// TIA Portal V16 export
// export: Created 2022-02-04T14:40:18.707467Z, ExportSetting WithDefaults, DisplayName Totally Integrated Automation Portal, DisplayVersion V16 Update 1, DisplayName TIA Portal Version Control Interface, DisplayVersion V16, DisplayName TIA Portal Openness, DisplayVersion V16, DisplayName SINAMICS Startdrive Advanced, DisplayVersion V16 Update 5, DisplayName SINAMICS Startdrive G130, G150, S120, S150, SINAMICS MV, S210, DisplayVersion V16 Update 5, DisplayName SINAMICS Startdrive G110M, G120, G120C, G120D, G120P, G115D, DisplayVersion V16 Update 5, DisplayName STEP 7 Professional, DisplayVersion V16, DisplayName STEP 7 Safety, DisplayVersion V16, DisplayName WinCC Advanced, DisplayVersion V16, DisplayName SIMATIC Visualization Architect, DisplayVersion V16
DATA_BLOCK "DGI"   // DB2
VERSION : 0.1
// stored: AutoNumber true, InstanceOfName GetDiskretInputs, InstanceOfType FB
"GetDiskretInputs"
   // VAR RETAIN
   //    K1_1122L1 : Bool;
   //    K1_113_13L1 : Bool;
   //    K1_113_24L1 : Bool;
   //    K1_113_35L1 : Bool;
   //    k1_113_46L1 : Bool;
   //    Varalla : Bool;
   //    Varalla1 : Bool;
   //    Varalla2 : Bool;
   //    F211K1_211K2 : Bool;
   //    F212K1 : Bool;
   //    F213K1 : Bool;
   //    F214K1 : Bool;
   //    Varalla3 : Bool;
   //    Varalla4 : Bool;
   //    Varalla5 : Bool;
   //    Varalla6 : Bool;
   //    F221K1 : Bool;
   //    F222K1 : Bool;
   //    F223K1 : Bool;
   //    F224K1 : Bool;
   //    F225K1 : Bool;
   //    F330K1 : Bool;
   //    Varalla8 : Bool;
   //    Varalla9 : Bool;
   //    F231K1 : Bool;
   //    F232K1 : Bool;
   //    F233K1 : Bool;
   //    F234K1 : Bool;
   //    F235K1_235K2 : Bool;
   //    Varalla10 : Bool;
   //    Varalla11 : Bool;
   //    Varalla12 : Bool;
   //    F311K1_311K2 : Bool;
   //    F312K1 : Bool;
   //    F313K1_313K2 : Bool;
   //    F314K1 : Bool;
   //    F315K1 : Bool;
   //    F316K1 : Bool;
   //    F317K1 : Bool;
   //    Varalla13 : Bool;
   //    F321K1_321K2 : Bool;
   //    F322K1_322K2 : Bool;
   //    F323K1_323K2 : Bool;
   //    F325K1 : Bool;
   //    Varalla14 : Bool;
   //    Varalla15 : Bool;
   //    Varalla16 : Bool;
   //    Varalla17 : Bool;
   //    F331K1 : Bool;
   //    F332K1 : Bool;
   //    F333K1 : Bool;
   //    F334K1 : Bool;
   //    F335K1 : Bool;
   //    F336K1 : Bool;
   //    F337K1 : Bool;
   //    K1_323U1 : Bool;
   //    K1_221U1 : Bool;
   //    K1_213U1 : Bool;
   //    K1_215U1 : Bool;
   //    K1_222U1 : Bool;
   //    K1_225U1 : Bool;
   //    K1_231U1 : Bool;
   //    K1_233U1 : Bool;
   //    K1_317U1 : Bool;
   //    K1_332U1 : Bool;
   //    K1_333U1 : Bool;
   //    K1_334U1 : Bool;
   //    K1_335U1 : Bool;
   //    K1_336U1 : Bool;
   //    K1_223U1 : Bool;
   //    K1_324U1 : Bool;
   //    K1_325U1 : Bool;
   //    K1_112_S1 : Bool;
   //    K1_112_S2 : Bool;
   //    K1_112_S3 : Bool;
   //    Varalla22 : Bool;
   //    K1_113_S11 : Bool;
   //    K1_113_S12 : Bool;
   //    k1_113_S13 : Bool;
   //    Varalla23 : Bool;
   //    Varalla24 : Bool;
   //    FC_223_1 : Bool;
   //    FC_223_2 : Bool;
   //    FC_223_3 : Bool;
   //    Varalla28 : Bool;
   //    Varalla29 : Bool;
   //    Varalla30 : Bool;
   //    Varalla31 : Bool;
   //    Liftdown : Bool;
   //    LiftUp : Bool;
   //    sloidoski : Bool;
   //    sloidoski2 : Bool;
   //    doskavpriymkeelevator : Bool;
   //    koncevik1 : Bool;
   //    koncevik2 : Bool;
   //    nakloniytransporter : Bool;
   //    FC_18_Length : Bool;
   //    F2_1m : Bool;
   //    F2_4m : Bool;
   //    F2_7m : Bool;
   //    F3_0m : Bool;
   //    F3_3m : Bool;
   //    F3_6m : Bool;
   //    F3_9m : Bool;
   //    F4_2m : Bool;
   //    F4_5m : Bool;
   //    F4_8m : Bool;
   //    F5_1m : Bool;
   //    F5_4m : Bool;
   //    F5_7m : Bool;
   //    F6_0m : Bool;
   //    PodBort_1 : Bool;
   //    PodBort_2 : Bool;
   //    "312Alarm" : Bool;
   //    S14_2 : Bool;
   //    S14_3 : Bool;
   //    B14_4 : Bool;
   //    B14_5 : Bool;
   //    K1_312U1 : Bool;
   //    S14_7 : Bool;
   //    S15_0 : Bool;
   //    S15_1 : Bool;
   //    S15_2 : Bool;
   //    reserv5 : Bool;
   //    Index : Bool;
   //    B15_5 : Bool;
   //    B15_6 : Bool;
   //    B15_7 : Bool;
   //    FC_232_1 : Bool;
   //    S16_1 : Bool;
   //    S16_2 : Bool;
   //    E16_3 : Bool;
   //    E16_4 : Bool;
   //    FC_232_2 : Bool;
   //    B16_6 : Bool;
   //    S16_7 : Bool;
   //    B17_0 : Bool;
   //    B17_1 : Bool;
   //    B17_2 : Bool;
   //    B17_3 : Bool;
   //    B17_4 : Bool;
   //    Varalla32 : Bool;
   //    Varalla33 : Bool;
   //    Varalla34 : Bool;
   //    B18_0 : Bool;
   //    B18_1 : Bool;
   //    S18_2 : Bool;
   //    S18_3 : Bool;
   //    B18_4 : Bool;
   //    B18_5 : Bool;
   //    B18_6 : Bool;
   //    B18_7 : Bool;
   //    B19_0 : Bool;
   //    Varalla35 : Bool;
   //    Varalla36 : Bool;
   //    Varalla37 : Bool;
   //    Varalla38 : Bool;
   //    Varalla39 : Bool;
   //    Varalla40 : Bool;
   //    Varalla41 : Bool;
   //    Varalla42 : Bool;
   //    Varalla43 : Bool;
   //    Varalla44 : Bool;
   //    Varalla45 : Bool;
   //    Varalla46 : Bool;
   //    Varalla47 : Bool;
   //    Varalla48 : Bool;
   //    Varalla49 : Bool;
   //    Varalla50 : Bool;
   //    Varalla51 : Bool;
   //    Varalla52 : Bool;
   //    Varalla53 : Bool;
   //    Varalla54 : Bool;
   //    Varalla55 : Bool;
   //    Varalla56 : Bool;
   //    Varalla57 : Bool;
   //    B22_0 : Bool;
   //    B22_1 : Bool;
   //    S22_2 : Bool;
   //    S22_3 : Bool;
   //    B22_4 : Bool;
   //    B22_5 : Bool;
   //    B22_6 : Bool;
   //    FC_22_7 : Bool;
   //    B23_0 : Bool;
   //    B23_1 : Bool;
   //    Varalla59 : Bool;
   //    Varalla60 : Bool;
   //    Varalla61 : Bool;
   //    Varalla62 : Bool;
   //    FC_23_6 : Bool;
   //    FC_23_7 : Bool;
   //    S76 : Bool;
   //    S76_1 : Bool;
   //    S76_2 : Bool;
   //    S76_3 : Bool;
   //    E76_4 : Bool;
   //    S76_5 : Bool;
   //    S76_6 : Bool;
   //    E76_7 : Bool;
   //    S77_0 : Bool;
   //    E77_1 : Bool;
   //    S77_2 : Bool;
   //    S77_3 : Bool;
   //    S77_4 : Bool;
   //    S77_5 : Bool;
   //    S77_6 : Bool;
   //    E77_7 : Bool;
   //    S78_0 : Bool;
   //    E78_1 : Bool;
   //    S78_2 : Bool;
   //    E78_3 : Bool;
   //    S78_4 : Bool;
   //    E78_5 : Bool;
   //    S78_6 : Bool;
   //    E78_7 : Bool;
   //    S79_0 : Bool;
   //    S79_1 : Bool;
   //    E79_2 : Bool;
   //    S79_3 : Bool;
   //    S79_4 : Bool;
   //    S79_5 : Bool;
   //    S79_6 : Bool;
   //    E79_7 : Bool;
   //    S80_0 : Bool;
   //    E80_1 : Bool;
   //    S80_2 : Bool;
   //    E80_3 : Bool;
   //    S80_4 : Bool;
   //    S80_5 : Bool;
   //    E80_6 : Bool;
   //    S80_7 : Bool;
   //    Varalla106 : Bool;
   //    Varalla107 : Bool;
   //    Varalla108 : Bool;
   //    Varalla109 : Bool;
   //    Varalla110 : Bool;
   //    Varalla111 : Bool;
   //    Varalla112 : Bool;
   //    Varalla113 : Bool;
   //    S82_0 : Bool;
   //    S81_1 : Bool;
   //    E82_2 : Bool;
   //    S82_3 : Bool;
   //    S82_4 : Bool;
   //    E82_5 : Bool;
   //    S82_6 : Bool;
   //    E82_7 : Bool;
   //    S83_0 : Bool;
   //    E83_1 : Bool;
   //    E83_2 : Bool;
   //    E83_3 : Bool;
   //    S83_4 : Bool;
   //    Varalla114 : Bool;
   //    Varalla115 : Bool;
   //    Varalla116 : Bool;
   //    S84_0 : Bool;
   //    S84_1 : Bool;
   //    E84_2 : Bool;
   //    S84_3 : Bool;
   //    S84_4 : Bool;
   //    S84_5 : Bool;
   //    E84_6 : Bool;
   //    S84_7 : Bool;
   //    E85_0 : Bool;
   //    S85_1 : Bool;
   //    E85_2 : Bool;
   //    S85_3 : Bool;
   //    E85_4 : Bool;
   //    S85_5 : Bool;
   //    E85_6 : Bool;
   //    S85_7 : Bool;
   //    S86_0 : Bool;
   //    E86_1 : Bool;
   //    S86_2 : Bool;
   //    S86_3 : Bool;
   //    S86_4 : Bool;
   //    S86_5 : Bool;
   //    Varalla117 : Bool;
   //    Varalla118 : Bool;
   //    S87_0 : Bool;
   //    S87_1 : Bool;
   //    E87_2 : Bool;
   //    S87_3 : Bool;
   //    S87_4 : Bool;
   //    Varalla119 : Bool;
   //    Varalla120 : Bool;
   //    Varalla121 : Bool;
   //    S88_0 : Bool;
   //    K3_3 : Bool;
   //    S88_2 : Bool;
   //    E88_3 : Bool;
   //    S88_4 : Bool;
   //    S88_5 : Bool;
   //    E88_6 : Bool;
   //    S88_7 : Bool;
   //    S89_0 : Bool;
   //    S89_1 : Bool;
   //    S89_2 : Bool;
   //    S89_3 : Bool;
   //    Varalla122 : Bool;
   //    Varalla123 : Bool;
   //    Varalla124 : Bool;
   //    Varalla125 : Bool;
   //    S90_0 : Bool;
   //    S90_1 : Bool;
   //    S90_2 : Bool;
   //    Varalla126 : Bool;
   //    S90_4 : Bool;
   //    E90_5 : Bool;
   //    S90_6 : Bool;
   //    E90_7 : Bool;
   //    S91_0 : Bool;
   //    E91_1 : Bool;
   //    S91_2 : Bool;
   //    Varalla127 : Bool;
   //    Varalla128 : Bool;
   //    Varalla129 : Bool;
   //    Varalla130 : Bool;
   //    Varalla131 : Bool;
   //    S214 : Bool;
   //    BrakDroper_front : Bool;
   //    BrakDroppperBob_old : Bool;
   //    UporDefectivePFM_timer : TON;
   //    GasketRampSqueeze_timer { S7_SetPoint := 'True'} : TON;
   //    TopSig_timer { S7_SetPoint := 'True'} : TON;
   //    PFMdefect_vill_fwd { S7_SetPoint := 'True'} : TON;
   //    MidSig_timer { S7_SetPoint := 'True'} : TOF;
   //    SensHook_timer { S7_SetPoint := 'True'} : TOF;
   //    SensHookDovod_timer { S7_SetPoint := 'True'} : TOF;
   //    SensStartEvalZone_timer { S7_SetPoint := 'True'} : TOF;
   //    SensEndEvalZone_timer { S7_SetPoint := 'True'} : TON;
   //    SensDropDefect_timer { S7_SetPoint := 'True'} : TOF;
   //    SensBoardCounter_timer { S7_SetPoint := 'True'} : TOF;
   //    SensBoardCounterFilter_timer { S7_SetPoint := 'True'} : TON;
   //    SensNewBobBrak_timer { S7_SetPoint := 'True'} : TOF;
   //    btn_Drop_Defect : "Button_ShortTap";
   //    "btn_Stop_M331/330" { S7_SetPoint := 'True'} : "Button_ShortTap";
   //    btn_btnLenta_defect { S7_SetPoint := 'True'} : "Button_ShortTap";
   //    btn_Force_Finish { S7_SetPoint := 'True'} : "Button_ShortTap";
   //    btn_DropFromRollerDefect { S7_SetPoint := 'True'} : "Button_ShortTap";
   //    btn_Cnrl_Mov_Side : "ButtonSwitcher_PlusLongTap";
   //    btn_Auto_Loading { S7_SetPoint := 'True'} : "ButtonSwitcher";
   //    btn_Auto_Sorting { S7_SetPoint := 'True'} : "ButtonSwitcher";
   //    btn_Auto_Gasket { S7_SetPoint := 'True'} : "ButtonSwitcher";
   //    btn_Auto_PFM_defective { S7_SetPoint := 'True'} : "ButtonSwitcher";
   //    btn_Reset_OP3 { S7_SetPoint := 'True'} : "ButtonShortLongTap";
   //    btn_ResetUporLine { S7_SetPoint := 'True'} : "Button_PlusLongTap";
   // END_VAR
BEGIN
END_DATA_BLOCK
